(* CoDeSys 2.3 export: TO_MIN.EXP *)

(* POU FUNv1/TO_MIN, ST *)
FUNCTION TO_MIN : TIME
VAR_INPUT
	in: DWORD;
END_VAR
VAR
END_VAR
TO_MIN := DWORD_TO_TIME(in)*60000;
END_FUNCTION
